REGION Network 77 (SCL): OPENVALVE
   IF ("MODE SELECTION DB"."MODE BUFF" <> 0 AND "TRANSFER DB".BUFF."MFG TO STORAGE-3 WITH INLINE FILTER PRES" = 2
       AND NOT "TRANSFER DB".PAUSE."MFG TO STORAGE-3 WITH INLINE FILTER PRES"
       AND "CONTINUE DB"."SYRUP MFG PROCESS ERROR" = 0 AND "LEVEL BUFF"."SYRUP MFG_LOAD CELL" = 0)
       OR ("MODE SELECTION DB"."MODE BUFF"=1 AND "MFG PROCESS_DB"."AUTO BUFF"=0
       AND "MFG TRANSFER CYCLE DB".TRANSFER."TRANSFER BUFF"."MFG TO STORAGE-3 WITH INLINE FILTER PRES"=10 AND "CONTINUE DB"."SYRUP MFG PROCESS ERROR" <>1
       AND "MFG TRANSFER CYCLE DB".TRANSFER.SELECT."SELECT BUFF"=6)
   THEN
       "TRANSFER DB".BIT."MFG TO STORAGE-3 WITH INLINE FILTER PRES"."PFBV-59 TANK OUTLET VALVE" := TRUE;
       "TRANSFER DB".BIT."MFG TO STORAGE-3 WITH INLINE FILTER PRES"."PBV-114 TANK OUTLET TO INLINE HOMOGENIZER LINE" := TRUE;
       "TRANSFER DB".BIT."MFG TO STORAGE-3 WITH INLINE FILTER PRES"."PBV-108 INLINE HOMOGENIZER TO FILTER PRESS INLET LINE" := TRUE;
       "TRANSFER DB".BIT."MFG TO STORAGE-3 WITH INLINE FILTER PRES"."FILTER PRESS MOTOR 1 RUN" := TRUE;
       "TRANSFER DB".BIT."MFG TO STORAGE-3 WITH INLINE FILTER PRES"."PBV-118 FILTER PRESS INLET" := TRUE;
       "TRANSFER DB".BIT."MFG TO STORAGE-3 WITH INLINE FILTER PRES"."PBV-111 FILTER PRESS OUTLER VALVE" := TRUE;
       "TRANSFER DB".BIT."MFG TO STORAGE-3 WITH INLINE FILTER PRES"."PBV-112 FILTER PRESS TO TRANSFER LINE" := TRUE;
       "TRANSFER DB".BIT."MFG TO STORAGE-3 WITH INLINE FILTER PRES"."PBV-117 MFG TO STORAGE – 3 TRANSFER LINE" := TRUE;
   ELSE
       "TRANSFER DB".BIT."MFG TO STORAGE-3 WITH INLINE FILTER PRES"."PFBV-59 TANK OUTLET VALVE" := FALSE;
       "TRANSFER DB".BIT."MFG TO STORAGE-3 WITH INLINE FILTER PRES"."PBV-114 TANK OUTLET TO INLINE HOMOGENIZER LINE" := FALSE;
       "TRANSFER DB".BIT."MFG TO STORAGE-3 WITH INLINE FILTER PRES"."PBV-108 INLINE HOMOGENIZER TO FILTER PRESS INLET LINE" := FALSE;
       "TRANSFER DB".BIT."MFG TO STORAGE-3 WITH INLINE FILTER PRES"."FILTER PRESS MOTOR 1 RUN" := FALSE;
       "TRANSFER DB".BIT."MFG TO STORAGE-3 WITH INLINE FILTER PRES"."PBV-118 FILTER PRESS INLET" := FALSE;
       "TRANSFER DB".BIT."MFG TO STORAGE-3 WITH INLINE FILTER PRES"."PBV-111 FILTER PRESS OUTLER VALVE" := FALSE;
       "TRANSFER DB".BIT."MFG TO STORAGE-3 WITH INLINE FILTER PRES"."PBV-112 FILTER PRESS TO TRANSFER LINE" := FALSE;
       "TRANSFER DB".BIT."MFG TO STORAGE-3 WITH INLINE FILTER PRES"."PBV-117 MFG TO STORAGE – 3 TRANSFER LINE" := FALSE;
       ;
   END_IF;
END_REGION

REGION Network 78: LOAD CELL_CUTOFF
   RUNG wire#powerrail
      { S7_Templates := "SrcType := Int" } NE_Contact(in1 := "MODE SELECTION DB"."MODE BUFF", in2 := 0)
      { S7_Templates := "SrcType := Int" } EQ_Contact(in1 := "TRANSFER DB".BUFF."MFG TO STORAGE-3 WITH INLINE FILTER PRES", in2 := 2)
      I_Contact( "TRANSFER DB".PAUSE."MFG TO STORAGE-3 WITH INLINE FILTER PRES" )
      { S7_Templates := "SrcType := Int" } NE_Contact(in1 := "CONTINUE DB"."SYRUP MFG PROCESS ERROR", in2 := 1)
      { S7_Templates := "SrcType := Int" } EQ_Contact(in1 := "LEVEL BUFF"."SYRUP MFG_LOAD CELL", in2 := 1)
      Move(in := 3, out1 => "TRANSFER DB".BUFF."MFG TO STORAGE-3 WITH INLINE FILTER PRES")
   END_RUNG
   // the same network as SCL:
   IF ("MODE SELECTION DB"."MODE BUFF" <> 0) AND ("TRANSFER DB".BUFF."MFG TO STORAGE-3 WITH INLINE FILTER PRES" = 2) AND NOT "TRANSFER DB".PAUSE."MFG TO STORAGE-3 WITH INLINE FILTER PRES" AND ("CONTINUE DB"."SYRUP MFG PROCESS ERROR" <> 1) AND ("LEVEL BUFF"."SYRUP MFG_LOAD CELL" = 1) THEN
       "TRANSFER DB".BUFF."MFG TO STORAGE-3 WITH INLINE FILTER PRES" := 3;
   END_IF;
END_REGION

REGION Network 79: PROCESS OVER & STOP
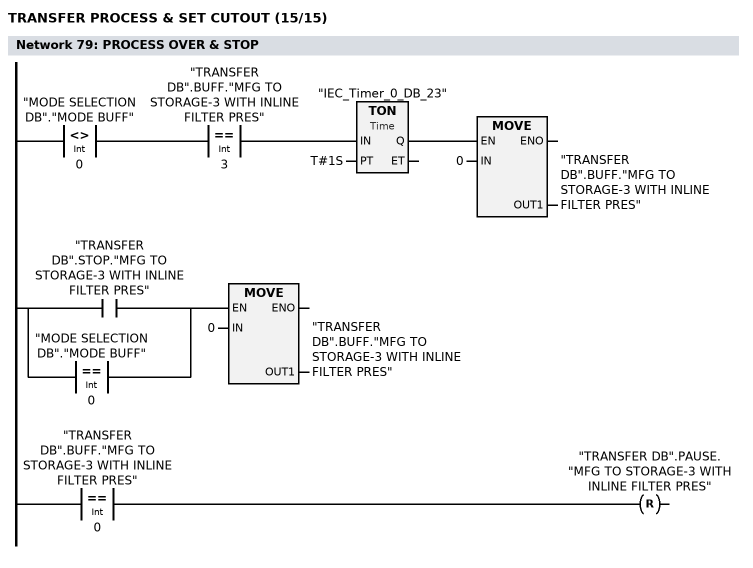
   RUNG wire#powerrail
      { S7_Templates := "SrcType := Int" } NE_Contact(in1 := "MODE SELECTION DB"."MODE BUFF", in2 := 0)
      { S7_Templates := "SrcType := Int" } EQ_Contact(in1 := "TRANSFER DB".BUFF."MFG TO STORAGE-3 WITH INLINE FILTER PRES", in2 := 3)
      { S7_Templates := "time_type := Time" } "IEC_Timer_0_DB_23".TON(pt := T#1S, et =>)
      Move(in := 0, out1 => "TRANSFER DB".BUFF."MFG TO STORAGE-3 WITH INLINE FILTER PRES")
   END_RUNG
   RUNG wire#powerrail
      Contact( "TRANSFER DB".STOP."MFG TO STORAGE-3 WITH INLINE FILTER PRES" )
      wire#w1
      Move(in := 0, out1 => "TRANSFER DB".BUFF."MFG TO STORAGE-3 WITH INLINE FILTER PRES")
   END_RUNG
   RUNG wire#powerrail
      { S7_Templates := "SrcType := Int" } EQ_Contact(in1 := "MODE SELECTION DB"."MODE BUFF", in2 := 0)
   END_RUNG wire#w1
   RUNG wire#powerrail
      { S7_Templates := "SrcType := Int" } EQ_Contact(in1 := "TRANSFER DB".BUFF."MFG TO STORAGE-3 WITH INLINE FILTER PRES", in2 := 0)
      R_Coil( "TRANSFER DB".PAUSE."MFG TO STORAGE-3 WITH INLINE FILTER PRES" )
   END_RUNG
   // the same network as SCL:
   "IEC_Timer_0_DB_23".TON(IN := ("MODE SELECTION DB"."MODE BUFF" <> 0) AND ("TRANSFER DB".BUFF."MFG TO STORAGE-3 WITH INLINE FILTER PRES" = 3),
                           PT := T#1S);
   IF "IEC_Timer_0_DB_23".Q THEN "TRANSFER DB".BUFF."MFG TO STORAGE-3 WITH INLINE FILTER PRES" := 0; END_IF;
   IF "TRANSFER DB".STOP."MFG TO STORAGE-3 WITH INLINE FILTER PRES" OR ("MODE SELECTION DB"."MODE BUFF" = 0) THEN
       "TRANSFER DB".BUFF."MFG TO STORAGE-3 WITH INLINE FILTER PRES" := 0;
   END_IF;
   IF "TRANSFER DB".BUFF."MFG TO STORAGE-3 WITH INLINE FILTER PRES" = 0 THEN
       "TRANSFER DB".PAUSE."MFG TO STORAGE-3 WITH INLINE FILTER PRES" := FALSE;
   END_IF;
END_REGION
END_FUNCTION
